TYPE "MotorAlr"
VERSION : 0.1
// Block: MotorAlr
   STRUCT
      ThermalProtection : Bool;
      Feedback : Bool;
   END_STRUCT;

END_TYPE
